DATA_BLOCK "PartData_Interface_DB"
VAR
  PartDataID : Int;
  PartData : Array[1..4] of "PartData_UDT";
  PartCMD : Array[1..4] of Struct;
END_VAR
BEGIN
END_DATA_BLOCK
